(* PLC project Untitled1, Beckhoff Automation GmbH TwinCAT PLC Control 3.5.13.20 *)
(* stored: creationDateTime 2022-07-20T15:22:52.6492138, modificationDateTime 2022-07-20T15:22:52.6492138 *)

{attribute 'qualified_only'}
{attribute 'strict'}
TYPE eFirmerOperatingState : (eNoInfo := 0, eOff := 1, eSleeping := 2, eStarting := 3, eMppt := 4, eThrottled := 5, eShuttingDown := 6, eFault := 7, eStandby := 8);
END_TYPE
